Fanuc KAREL source: kt00345.KL

-- PROVISIONAL review KL for V1013-1; original PC SHA256 491d339efa0889fee49680b1f1eb94e79c932c665cfb97d11daada41a512618d
-- Incomplete behavior may be omitted. Consult companion uncertainty JSON. Do not deploy.
PROGRAM KT00345
%NOLOCKGROUP
VAR
  OUT : BOOLEAN
-- UNRESOLVED_DECL H1 type=002017
-- UNRESOLVED_DECL Y2 type=002018
BEGIN
  -- UNRESOLVED_PC offsets 5-19; opcodes 2E,22,9D,33,B4
  -- UNRESOLVED_PC offsets 24-38; opcodes 2E,22,9D,33,B2
  -- UNRESOLVED_PC offsets 43-68; opcodes 22,9D,33,B3,22,9D,33,B1,59,23
  -- UNRESOLVED_PC offsets 73-77; opcodes 7F
END KT00345
